// TIA Portal V20 export
VAR_GLOBAL   // PLC tag table "Constantes de Eventos AGenerar"
END_VAR
VAR_GLOBAL CONSTANT   // user constants
   Evento_VTDC_PosicionActualVTD : UInt := 650;
   Evento_DISPOSITIVO_EstadoActual : UInt := 160;
   Evento_DISPOSITIVO_FinReset_OK : UInt := 151;
   Evento_DISPOSITIVO_FinReset_NOK : UInt := 152;
   Evento_DISPOSITIVO_FinParoBlando_OK : UInt := 153;
   Evento_DISPOSITIVO_FinParoBlando_NOK : UInt := 154;
   Evento_VTDC_FinPosicionado_OK : UInt := 660;
   Evento_VTDC_FinPosicionado_NOK : UInt := 661;
END_VAR
